// TIA Portal project "WaterFiltering" (V15)

(* hardware
DEVICE "S7-1200 station_1"  S7-1200 Station
   slot 0: "Rack_0"  S7-1200 Rack  Rack  V1.0
   slot 1: "PLC_1"  CPU 1214C AC/DC/Rly  6ES7 214-1BG40-0XB0  V4.2
DEVICE "PC-System_1"  SIMATIC PC station
   slot 0: "SIMATIC PC station"  Rail  SIMATIC PC-Station  V1.0
      slot 125: "Stationmanager"  Station_Manager  V6.0.4
   slot 1: "HMI_RT_1"  WinCC RT Professional  6AV2 105-0xxxx-xxxx  15.0.0.0
   slot 2: "IE general_1"  IE General  IE_CP  V8.2.0
*)

// ===== PLC "PLC_1"  CPU 1214C AC/DC/Rly =====

VAR_GLOBAL   // PLC tag table "Default tag table"
   "FlowSwitch" AT %M0.0 : Bool;
   "PressureInput2" AT %MW0 : Int;
   "PressureInput1" AT %MW2 : Int;
   "ScaledPressure1" AT %MW4 : Int;
   "ScaledPressure2" AT %MW6 : Int;
   "DifferPressureRaw" AT %MW8 : Int;
   "DifferPressure" AT %MW10 : Int;
   "LevelInput" AT %MW12 : Int;
   "ScaledLevel" AT %MW14 : Int;
   "SV1Off_Pb" AT %M16.0 : Bool;
   "SV1Hand_Pb" AT %M16.1 : Bool;
   "SV1Auto_Pb" AT %M16.2 : Bool;
   "SV2Off_Pb" AT %M16.3 : Bool;
   "SV2Hand_Pb" AT %M16.4 : Bool;
   "SV2Auto_pb" AT %M16.5 : Bool;
   "SV3Off_pb" AT %M16.6 : Bool;
   "SV3Hand_pb" AT %M16.7 : Bool;
   "SV3Auto_Pb" AT %M17.0 : Bool;
   "SV4Off_pb" AT %M17.1 : Bool;
   "SV4Hand_Pb" AT %M17.2 : Bool;
   "SV4Auto_Pb" AT %M17.3 : Bool;
   "SV5Off_Pb" AT %M17.4 : Bool;
   "SV5Hand_Pb" AT %M17.5 : Bool;
   "SV5Auto_Pb" AT %M17.6 : Bool;
   "SV6Off_Pb" AT %M17.7 : Bool;
   "SV6Hand_Pb" AT %M18.0 : Bool;
   "SV6Auto_pb" AT %M18.1 : Bool;
   "SV1_Status" AT %MW18 : Int;
   "SV2_Status" AT %MW20 : Int;
   "SV3_Status" AT %MW22 : Int;
   "SV4_Status" AT %MW24 : Int;
   "SV5_Status" AT %MW26 : Int;
   "SV6_Status" AT %MW28 : Int;
   "PumpOff_pb" AT %M2.0 : Bool;
   "PumpHand_pb" AT %M2.1 : Bool;
   "PumpAuto_pb" AT %M2.2 : Bool;
   "Pump_Status" AT %MW30 : Int;
   "AllHOAAuto" AT %M32.0 : Bool;
   "Sys_Running" AT %M32.3 : Bool;
   "Critical_Alarm" AT %M32.6 : Bool;
   "BackWash_Running" AT %M32.7 : Bool;
   "Tank_Filling" AT %M39.0 : Bool;
   "FillStart_Trigger" AT %M33.7 : Bool;
   "FillStop_Trigger" AT %M34.0 : Bool;
   "Alarm_Reset" AT %M34.1 : Bool;
   "HiPresAlarm_Trigger" AT %M34.2 : Bool;
   "HiPres_Alarm" AT %M34.3 : Bool;
   "HiPres_Notify" AT %M34.4 : Bool;
   "Alarm_Silence" AT %M34.5 : Bool;
   "LowFlowAlm_Trigger" AT %M33.0 : Bool;
   "LowFlow_Alarm" AT %M33.1 : Bool;
   "LowAlarm_Notify" AT %M33.2 : Bool;
   "LowLevelAlm_Trigger" AT %M33.3 : Bool;
   "LowLevel_Alarm" AT %M33.4 : Bool;
   "LowLevelAlm_Notify" AT %M33.5 : Bool;
   "HighLevelAlm_Trigger" AT %M34.6 : Bool;
   "HighLevel_Alarm" AT %M34.7 : Bool;
   "HighLevelAlm_notify" AT %M35.0 : Bool;
   "BW_Lockout_Pb" AT %M35.1 : Bool;
   "BW_Lockout" AT %M35.2 : Bool;
   "BW_Enable_Pb" AT %M35.3 : Bool;
   "BWPending_Trigger" AT %M35.4 : Bool;
   "ManualBW_Pb" AT %M35.5 : Bool;
   "BWPending" AT %M35.6 : Bool;
   "BWCycle_Trigger" AT %M35.7 : Bool;
   "BWCount" AT %MW36 : Int;
   "ResetBW_Count_Pb" AT %M38.0 : Bool;
   "Filter_Resistance" AT %MW40 : Int;
   "LowFlowAlm_Pb" AT %M38.1 : Bool;
   "LowFlowAlm_pending" AT %M38.2 : Bool;
   "PutAllIntoAuto" AT %M38.3 : Bool;
   "JustCheck" AT %M38.4 : Bool;
   "St" AT %M38.7 : Bool;
   "FillStart_pulse" AT %M33.6 : Bool;
   "FillStop_Pulse" AT %M39.1 : Bool;
   "SysStart_Pb" AT %M32.1 : Bool;
   "SysStart_Trigger" AT %M32.4 : Bool;
   "SysStop_Pb" AT %M32.5 : Bool;
   "SysStop_Trigger" AT %M38.6 : Bool;
   "SolValve1" AT %Q0.0 : Bool;
   "SolValve2" AT %Q0.1 : Bool;
   "SolValve3" AT %Q0.2 : Bool;
   "SolValve4" AT %Q0.3 : Bool;
   "SolValve5" AT %Q0.4 : Bool;
   "SolValve6" AT %Q0.5 : Bool;
   "Pump" AT %Q0.6 : Bool;
END_VAR

DATA_BLOCK "ALARMS_DB"   // DB1
{ S7_Optimized_Access := 'TRUE' }
VERSION : 0.1
// stored: InstanceOfName ALARMS
"ALARMS"
BEGIN
END_DATA_BLOCK

DATA_BLOCK "MODE_DB"   // DB4
{ S7_Optimized_Access := 'TRUE' }
VERSION : 0.1
// stored: InstanceOfName MODE
"MODE"
BEGIN
END_DATA_BLOCK

DATA_BLOCK "ANALOG_DB"   // DB6
{ S7_Optimized_Access := 'TRUE' }
VERSION : 0.1
// stored: InstanceOfName ANALOG
"ANALOG"
BEGIN
END_DATA_BLOCK

DATA_BLOCK "SIM_DB"   // DB8
{ S7_Optimized_Access := 'TRUE' }
VERSION : 0.1
// stored: InstanceOfName SIM
"SIM"
BEGIN
END_DATA_BLOCK

DATA_BLOCK "LEVEL_DB"   // DB9
{ S7_Optimized_Access := 'TRUE' }
VERSION : 0.1
// stored: InstanceOfName LEVEL
"LEVEL"
BEGIN
END_DATA_BLOCK

DATA_BLOCK "BACKWASH_DB"   // DB10
{ S7_Optimized_Access := 'TRUE' }
VERSION : 0.1
// stored: InstanceOfName BACKWASH
"BACKWASH"
BEGIN
END_DATA_BLOCK

DATA_BLOCK "CTRL_DB"   // DB15
{ S7_Optimized_Access := 'TRUE' }
VERSION : 0.1
// stored: InstanceOfName CTRL
"CTRL"
BEGIN
END_DATA_BLOCK

DATA_BLOCK "HOA_DB"   // DB20
{ S7_Optimized_Access := 'TRUE' }
VERSION : 0.1
// stored: InstanceOfName HOA
"HOA"
BEGIN
END_DATA_BLOCK

DATA_BLOCK "REVIEW_DB"   // DB22
{ S7_Optimized_Access := 'TRUE' }
VERSION : 0.1
// stored: InstanceOfName REVIEW
"REVIEW"
BEGIN
END_DATA_BLOCK

// folder: System blocks/Program resources

DATA_BLOCK "HiPresAlm_Delay"   // DB2
{ S7_Optimized_Access := 'TRUE' }
AUTHOR : Simatic
FAMILY : IEC
NAME : IEC_TMR
VERSION : 1.0
// stored: InstanceOfName IEC_TIMER
"IEC_TIMER"
BEGIN
END_DATA_BLOCK

DATA_BLOCK "LowFlowAlm_Delay"   // DB3
{ S7_Optimized_Access := 'TRUE' }
AUTHOR : Simatic
FAMILY : IEC
NAME : IEC_TMR
VERSION : 1.0
// stored: InstanceOfName IEC_TIMER
"IEC_TIMER"
BEGIN
END_DATA_BLOCK

DATA_BLOCK "FillStart_Delay"   // DB5
{ S7_Optimized_Access := 'TRUE' }
AUTHOR : Simatic
FAMILY : IEC
NAME : IEC_TMR
VERSION : 1.0
// stored: InstanceOfName IEC_TIMER
"IEC_TIMER"
BEGIN
END_DATA_BLOCK

DATA_BLOCK "Simulation_Timer"   // DB7
{ S7_Optimized_Access := 'TRUE' }
AUTHOR : Simatic
FAMILY : IEC
NAME : IEC_TMR
VERSION : 1.0
// stored: InstanceOfName IEC_TIMER
"IEC_TIMER"
BEGIN
END_DATA_BLOCK

DATA_BLOCK "FillStop_Delay"   // DB11
{ S7_Optimized_Access := 'TRUE' }
AUTHOR : Simatic
FAMILY : IEC
NAME : IEC_TMR
VERSION : 1.0
// stored: InstanceOfName IEC_TIMER
"IEC_TIMER"
BEGIN
END_DATA_BLOCK

DATA_BLOCK "HiLevelAlm_Delay"   // DB13
{ S7_Optimized_Access := 'TRUE' }
AUTHOR : Simatic
FAMILY : IEC
NAME : IEC_TMR
VERSION : 1.0
// stored: InstanceOfName IEC_TIMER
"IEC_TIMER"
BEGIN
END_DATA_BLOCK

DATA_BLOCK "LowLevelAlm_Delay"   // DB14
{ S7_Optimized_Access := 'TRUE' }
AUTHOR : Simatic
FAMILY : IEC
NAME : IEC_TMR
VERSION : 1.0
// stored: InstanceOfName IEC_TIMER
"IEC_TIMER"
BEGIN
END_DATA_BLOCK

DATA_BLOCK "BWPending_Delay"   // DB16
{ S7_Optimized_Access := 'TRUE' }
AUTHOR : Simatic
FAMILY : IEC
NAME : IEC_TMR
VERSION : 1.0
// stored: InstanceOfName IEC_TIMER
"IEC_TIMER"
BEGIN
END_DATA_BLOCK

DATA_BLOCK "BWCycle_Delay"   // DB17
{ S7_Optimized_Access := 'TRUE' }
AUTHOR : Simatic
FAMILY : IEC
NAME : IEC_TMR
VERSION : 1.0
// stored: InstanceOfName IEC_TIMER
"IEC_TIMER"
BEGIN
END_DATA_BLOCK

DATA_BLOCK "BWCycle"   // DB18
{ S7_Optimized_Access := 'TRUE' }
AUTHOR : Simatic
FAMILY : IEC
NAME : IEC_TMR
VERSION : 1.0
// stored: InstanceOfName IEC_TIMER
"IEC_TIMER"
BEGIN
END_DATA_BLOCK

DATA_BLOCK "ResetBWCount_Delay"   // DB19
{ S7_Optimized_Access := 'TRUE' }
AUTHOR : Simatic
FAMILY : IEC
NAME : IEC_TMR
VERSION : 1.0
// stored: InstanceOfName IEC_TIMER
"IEC_TIMER"
BEGIN
END_DATA_BLOCK

DATA_BLOCK "FlowSWClose_Delay"   // DB21
{ S7_Optimized_Access := 'TRUE' }
AUTHOR : Simatic
FAMILY : IEC
NAME : IEC_TMR
VERSION : 1.0
// stored: InstanceOfName IEC_TIMER
"IEC_TIMER"
BEGIN
END_DATA_BLOCK

// folder: (top level)

FUNCTION_BLOCK "ANALOG"   // FB1, LAD
{ S7_Optimized_Access := 'TRUE' }
VERSION : 0.1
BEGIN

REGION Network 1
   // Analog Input : Pressure(0-20 psi), Water level(0-100)
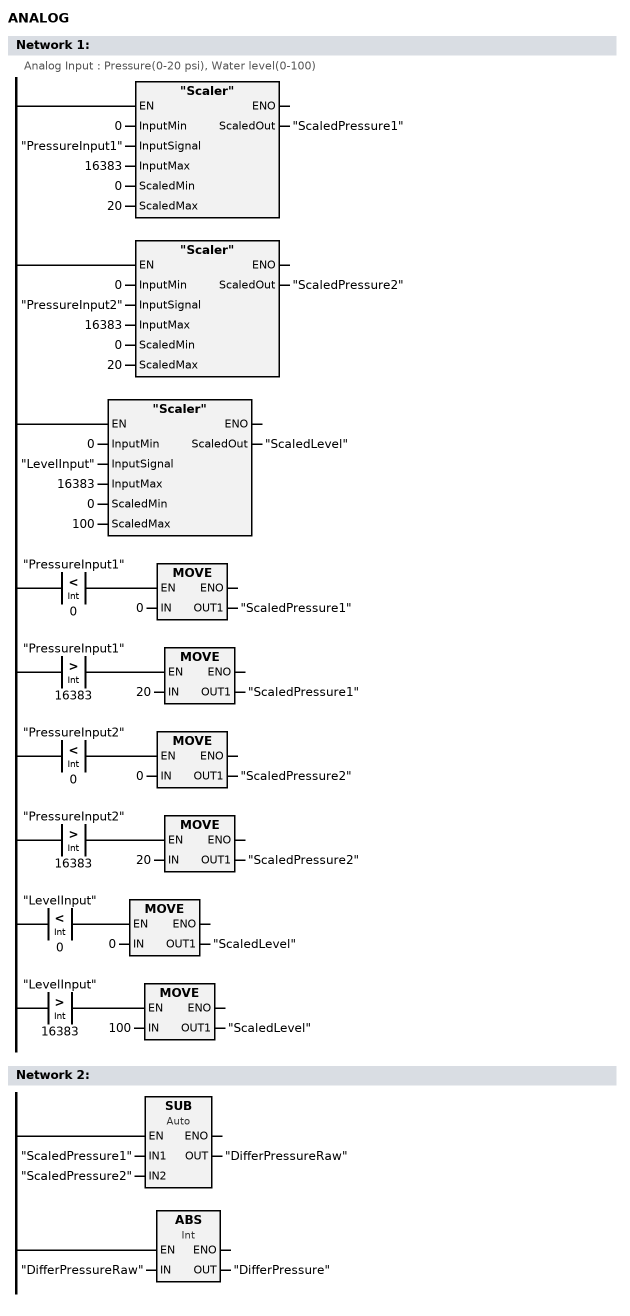
   RUNG wire#powerrail
      "Scaler"(InputMin := 0, InputSignal := "PressureInput1", InputMax := 16383, ScaledMin := 0, ScaledMax := 20, ScaledOut => "ScaledPressure1")
   END_RUNG
   RUNG wire#powerrail
      "Scaler"(InputMin := 0, InputSignal := "PressureInput2", InputMax := 16383, ScaledMin := 0, ScaledMax := 20, ScaledOut => "ScaledPressure2")
   END_RUNG
   RUNG wire#powerrail
      "Scaler"(InputMin := 0, InputSignal := "LevelInput", InputMax := 16383, ScaledMin := 0, ScaledMax := 100, ScaledOut => "ScaledLevel")
   END_RUNG
   RUNG wire#powerrail
      { S7_Templates := "SrcType := Int" } LT_Contact(in1 := "PressureInput1", in2 := 0)
      { S7_GenerateENO := "TRUE" } Move(in := 0, out1 => "ScaledPressure1")
   END_RUNG
   RUNG wire#powerrail
      { S7_Templates := "SrcType := Int" } GT_Contact(in1 := "PressureInput1", in2 := 16383)
      { S7_GenerateENO := "TRUE" } Move(in := 20, out1 => "ScaledPressure1")
   END_RUNG
   RUNG wire#powerrail
      { S7_Templates := "SrcType := Int" } LT_Contact(in1 := "PressureInput2", in2 := 0)
      { S7_GenerateENO := "TRUE" } Move(in := 0, out1 => "ScaledPressure2")
   END_RUNG
   RUNG wire#powerrail
      { S7_Templates := "SrcType := Int" } GT_Contact(in1 := "PressureInput2", in2 := 16383)
      { S7_GenerateENO := "TRUE" } Move(in := 20, out1 => "ScaledPressure2")
   END_RUNG
   RUNG wire#powerrail
      { S7_Templates := "SrcType := Int" } LT_Contact(in1 := "LevelInput", in2 := 0)
      { S7_GenerateENO := "TRUE" } Move(in := 0, out1 => "ScaledLevel")
   END_RUNG
   RUNG wire#powerrail
      { S7_Templates := "SrcType := Int" } GT_Contact(in1 := "LevelInput", in2 := 16383)
      { S7_GenerateENO := "TRUE" } Move(in := 100, out1 => "ScaledLevel")
   END_RUNG
   // the same network as SCL:
   "Scaler"(InputMin := 0,
            InputSignal := "PressureInput1",
            InputMax := 16383,
            ScaledMin := 0,
            ScaledMax := 20,
            ScaledOut => "ScaledPressure1");
   "Scaler"(InputMin := 0,
            InputSignal := "PressureInput2",
            InputMax := 16383,
            ScaledMin := 0,
            ScaledMax := 20,
            ScaledOut => "ScaledPressure2");
   "Scaler"(InputMin := 0,
            InputSignal := "LevelInput",
            InputMax := 16383,
            ScaledMin := 0,
            ScaledMax := 100,
            ScaledOut => "ScaledLevel");
   IF "PressureInput1" < 0 THEN "ScaledPressure1" := 0; END_IF;
   IF "PressureInput1" > 16383 THEN "ScaledPressure1" := 20; END_IF;
   IF "PressureInput2" < 0 THEN "ScaledPressure2" := 0; END_IF;
   IF "PressureInput2" > 16383 THEN "ScaledPressure2" := 20; END_IF;
   IF "LevelInput" < 0 THEN "ScaledLevel" := 0; END_IF;
   IF "LevelInput" > 16383 THEN "ScaledLevel" := 100; END_IF;
END_REGION

REGION Network 2
   RUNG wire#powerrail
      { S7_GenerateENO := "TRUE" } Sub(in1 := "ScaledPressure1", in2 := "ScaledPressure2", out => "DifferPressureRaw")
   END_RUNG
   RUNG wire#powerrail
      { S7_Templates := "SrcType := Int"; S7_GenerateENO := "TRUE" } Abs(in := "DifferPressureRaw", out => "DifferPressure")
   END_RUNG
   // the same network as SCL:
   "DifferPressureRaw" := "ScaledPressure1" - "ScaledPressure2";
   "DifferPressure" := ABS("DifferPressureRaw");
END_REGION
END_FUNCTION_BLOCK

FUNCTION_BLOCK "ALARMS"   // FB2, LAD
{ S7_Optimized_Access := 'TRUE' }
VERSION : 0.1
   VAR
      ons1 : Bool;
      ons2 : Bool;
      ons3 : Bool;
      ons4 : Bool;
   END_VAR
   VAR_TEMP   // added for the SCL form of the ladder/FBD networks
      _w1 : Bool;
   END_VAR
BEGIN

REGION Network 1
   // High Pressure Alarm
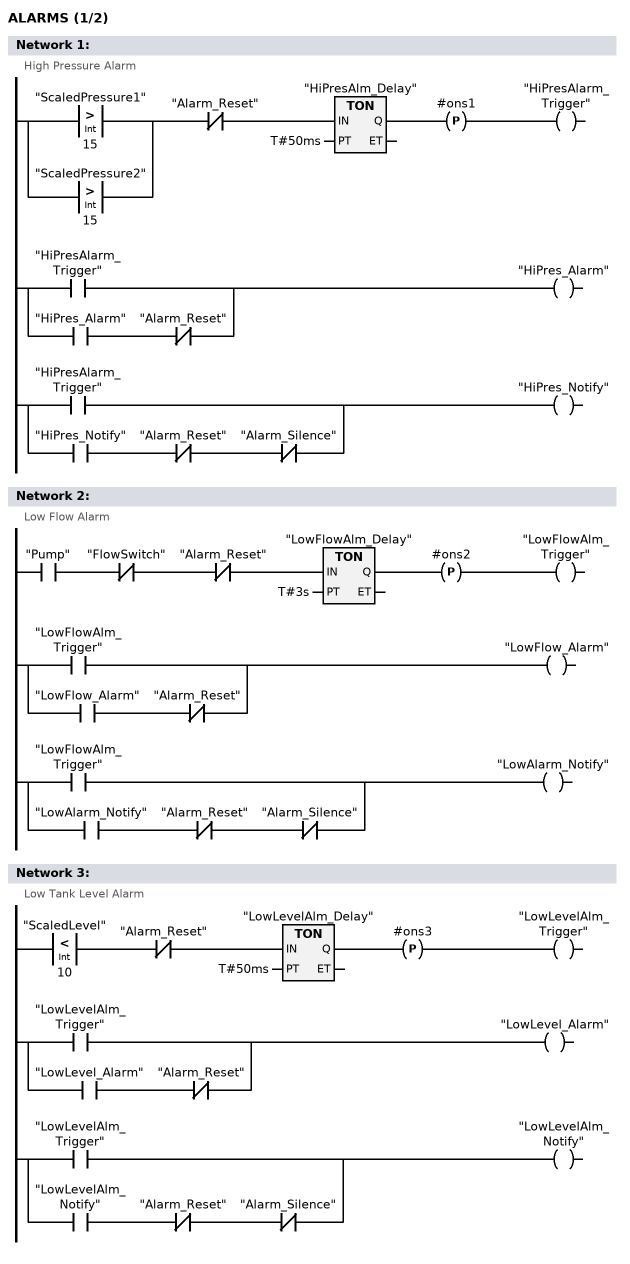
   "HiPresAlm_Delay".TON(IN := (("ScaledPressure1" > 15) OR ("ScaledPressure2" > 15)) AND NOT "Alarm_Reset",
                         PT := T#50ms);
   #_w1 := "HiPresAlm_Delay".Q AND NOT #ons1;   // rising edge
   #ons1 := "HiPresAlm_Delay".Q;
   "HiPresAlarm_Trigger" := #_w1;
   "HiPres_Alarm" := "HiPresAlarm_Trigger" OR ("HiPres_Alarm" AND NOT "Alarm_Reset");
   "HiPres_Notify" := "HiPresAlarm_Trigger" OR ("HiPres_Notify" AND NOT "Alarm_Reset" AND NOT "Alarm_Silence");
END_REGION

REGION Network 2
   // Low Flow Alarm
   "LowFlowAlm_Delay".TON(IN := "Pump" AND NOT "FlowSwitch" AND NOT "Alarm_Reset", PT := T#3s);
   #_w1 := "LowFlowAlm_Delay".Q AND NOT #ons2;   // rising edge
   #ons2 := "LowFlowAlm_Delay".Q;
   "LowFlowAlm_Trigger" := #_w1;
   "LowFlow_Alarm" := "LowFlowAlm_Trigger" OR ("LowFlow_Alarm" AND NOT "Alarm_Reset");
   "LowAlarm_Notify" := "LowFlowAlm_Trigger" OR ("LowAlarm_Notify" AND NOT "Alarm_Reset" AND NOT "Alarm_Silence");
END_REGION

REGION Network 3
   // Low Tank Level Alarm
   "LowLevelAlm_Delay".TON(IN := ("ScaledLevel" < 10) AND NOT "Alarm_Reset", PT := T#50ms);
   #_w1 := "LowLevelAlm_Delay".Q AND NOT #ons3;   // rising edge
   #ons3 := "LowLevelAlm_Delay".Q;
   "LowLevelAlm_Trigger" := #_w1;
   "LowLevel_Alarm" := "LowLevelAlm_Trigger" OR ("LowLevel_Alarm" AND NOT "Alarm_Reset");
   "LowLevelAlm_Notify" := "LowLevelAlm_Trigger" OR ("LowLevelAlm_Notify" AND NOT "Alarm_Reset" AND NOT "Alarm_Silence");
END_REGION

REGION Network 4
   // High Level Alarm
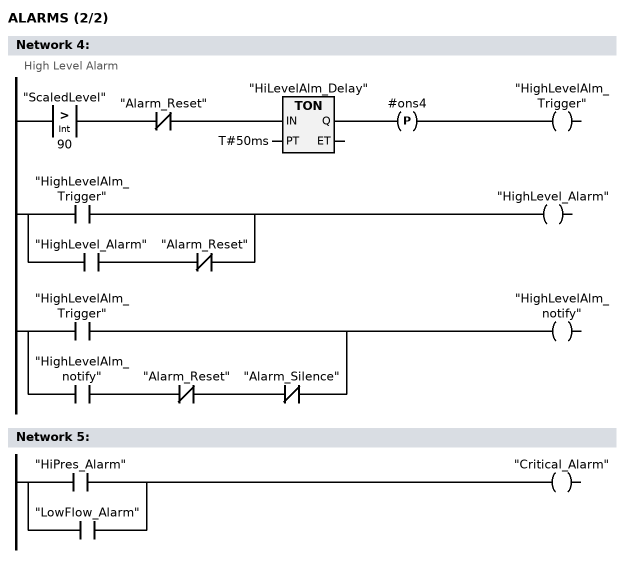
   "HiLevelAlm_Delay".TON(IN := ("ScaledLevel" > 90) AND NOT "Alarm_Reset", PT := T#50ms);
   #_w1 := "HiLevelAlm_Delay".Q AND NOT #ons4;   // rising edge
   #ons4 := "HiLevelAlm_Delay".Q;
   "HighLevelAlm_Trigger" := #_w1;
   "HighLevel_Alarm" := "HighLevelAlm_Trigger" OR ("HighLevel_Alarm" AND NOT "Alarm_Reset");
   "HighLevelAlm_notify" := "HighLevelAlm_Trigger" OR ("HighLevelAlm_notify" AND NOT "Alarm_Reset" AND NOT "Alarm_Silence");
END_REGION

REGION Network 5
   RUNG wire#powerrail
      Contact( "HiPres_Alarm" )
      wire#w1
      Coil( "Critical_Alarm" )
   END_RUNG
   RUNG wire#powerrail
      Contact( "LowFlow_Alarm" )
   END_RUNG wire#w1
   // the same network as SCL:
   "Critical_Alarm" := "HiPres_Alarm" OR "LowFlow_Alarm";
END_REGION
END_FUNCTION_BLOCK

FUNCTION_BLOCK "CTRL"   // FB3, LAD
{ S7_Optimized_Access := 'TRUE' }
VERSION : 0.1
BEGIN

REGION Network 1
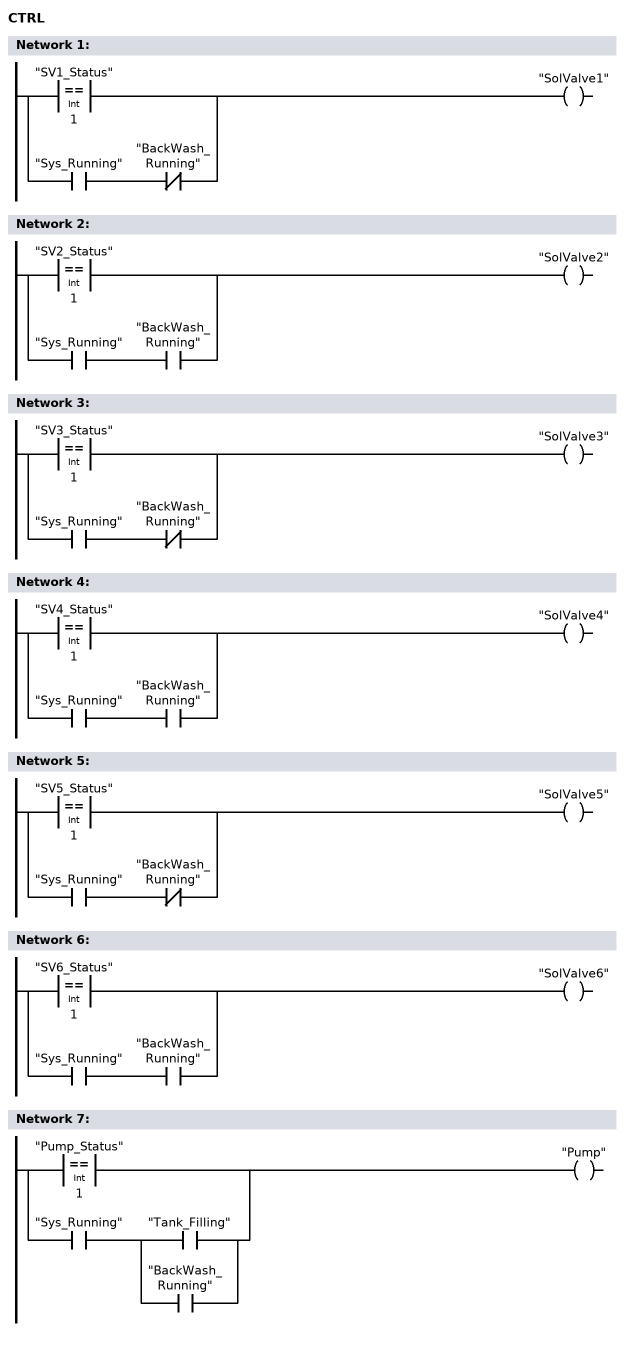
   RUNG wire#powerrail
      { S7_Templates := "SrcType := Int" } EQ_Contact(in1 := "SV1_Status", in2 := 1)
      wire#w1
      Coil( "SolValve1" )
   END_RUNG
   RUNG wire#powerrail
      Contact( "Sys_Running" )
      I_Contact( "BackWash_Running" )
   END_RUNG wire#w1
   // the same network as SCL:
   "SolValve1" := ("SV1_Status" = 1) OR ("Sys_Running" AND NOT "BackWash_Running");
END_REGION

REGION Network 2
   RUNG wire#powerrail
      { S7_Templates := "SrcType := Int" } EQ_Contact(in1 := "SV2_Status", in2 := 1)
      wire#w1
      Coil( "SolValve2" )
   END_RUNG
   RUNG wire#powerrail
      Contact( "Sys_Running" )
      Contact( "BackWash_Running" )
   END_RUNG wire#w1
   // the same network as SCL:
   "SolValve2" := ("SV2_Status" = 1) OR ("Sys_Running" AND "BackWash_Running");
END_REGION

REGION Network 3
   RUNG wire#powerrail
      { S7_Templates := "SrcType := Int" } EQ_Contact(in1 := "SV3_Status", in2 := 1)
      wire#w1
      Coil( "SolValve3" )
   END_RUNG
   RUNG wire#powerrail
      Contact( "Sys_Running" )
      I_Contact( "BackWash_Running" )
   END_RUNG wire#w1
   // the same network as SCL:
   "SolValve3" := ("SV3_Status" = 1) OR ("Sys_Running" AND NOT "BackWash_Running");
END_REGION

REGION Network 4
   RUNG wire#powerrail
      { S7_Templates := "SrcType := Int" } EQ_Contact(in1 := "SV4_Status", in2 := 1)
      wire#w1
      Coil( "SolValve4" )
   END_RUNG
   RUNG wire#powerrail
      Contact( "Sys_Running" )
      Contact( "BackWash_Running" )
   END_RUNG wire#w1
   // the same network as SCL:
   "SolValve4" := ("SV4_Status" = 1) OR ("Sys_Running" AND "BackWash_Running");
END_REGION

REGION Network 5
   RUNG wire#powerrail
      { S7_Templates := "SrcType := Int" } EQ_Contact(in1 := "SV5_Status", in2 := 1)
      wire#w1
      Coil( "SolValve5" )
   END_RUNG
   RUNG wire#powerrail
      Contact( "Sys_Running" )
      I_Contact( "BackWash_Running" )
   END_RUNG wire#w1
   // the same network as SCL:
   "SolValve5" := ("SV5_Status" = 1) OR ("Sys_Running" AND NOT "BackWash_Running");
END_REGION

REGION Network 6
   RUNG wire#powerrail
      { S7_Templates := "SrcType := Int" } EQ_Contact(in1 := "SV6_Status", in2 := 1)
      wire#w1
      Coil( "SolValve6" )
   END_RUNG
   RUNG wire#powerrail
      Contact( "Sys_Running" )
      Contact( "BackWash_Running" )
   END_RUNG wire#w1
   // the same network as SCL:
   "SolValve6" := ("SV6_Status" = 1) OR ("Sys_Running" AND "BackWash_Running");
END_REGION

REGION Network 7
   RUNG wire#powerrail
      { S7_Templates := "SrcType := Int" } EQ_Contact(in1 := "Pump_Status", in2 := 1)
      wire#w1
      Coil( "Pump" )
   END_RUNG
   RUNG wire#powerrail
      Contact( "Sys_Running" )
      wire#w2
      Contact( "Tank_Filling" )
   END_RUNG wire#w1
   RUNG wire#w2
      Contact( "BackWash_Running" )
   END_RUNG wire#w1
   // the same network as SCL:
   "Pump" := ("Pump_Status" = 1) OR ("Sys_Running" AND ("Tank_Filling" OR "BackWash_Running"));
END_REGION
END_FUNCTION_BLOCK

FUNCTION_BLOCK "HOA"   // FB4, LAD
{ S7_Optimized_Access := 'TRUE' }
VERSION : 0.1
   VAR
      ons1 : Bool;
      ons2 : Bool;
      ons3 : Bool;
      ons4 : Bool;
      ons5 : Bool;
      ons6 : Bool;
      ons7 : Bool;
      ons8 : Bool;
      ons9 : Bool;
      ons10 : Bool;
      ons11 : Bool;
      ons12 : Bool;
      ons13 : Bool;
      ons14 : Bool;
      ons15 : Bool;
      ons16 : Bool;
      ons17 : Bool;
      ons18 : Bool;
      ons19 : Bool;
      ons20 : Bool;
      ons21 : Bool;
   END_VAR
   VAR_TEMP   // added for the SCL form of the ladder/FBD networks
      _w1 : Bool;
      _w2 : Bool;
      _w3 : Bool;
   END_VAR
BEGIN

REGION Network 1
   // Solenoid Valve1 HOA
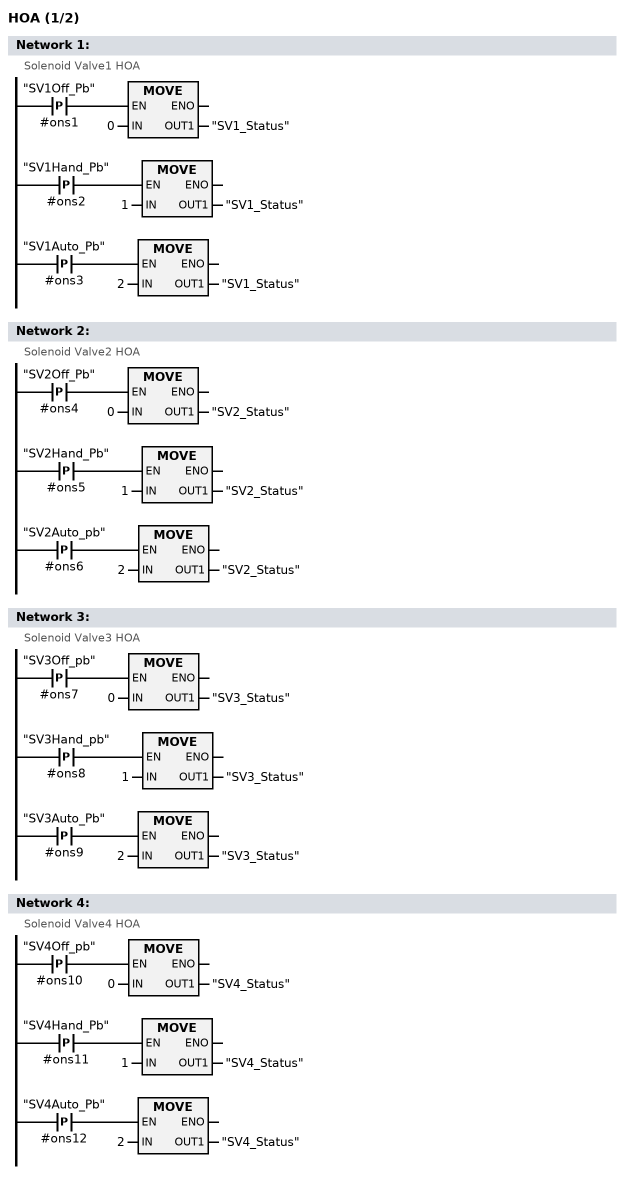
   RUNG wire#powerrail
      P_Contact(operand := "SV1Off_Pb", bit := #ons1)
      { S7_GenerateENO := "TRUE" } Move(in := 0, out1 => "SV1_Status")
   END_RUNG
   RUNG wire#powerrail
      P_Contact(operand := "SV1Hand_Pb", bit := #ons2)
      { S7_GenerateENO := "TRUE" } Move(in := 1, out1 => "SV1_Status")
   END_RUNG
   RUNG wire#powerrail
      P_Contact(operand := "SV1Auto_Pb", bit := #ons3)
      { S7_GenerateENO := "TRUE" } Move(in := 2, out1 => "SV1_Status")
   END_RUNG
   // the same network as SCL:
   #_w1 := "SV1Off_Pb" AND NOT #ons1;   // rising edge of "SV1Off_Pb"
   #ons1 := "SV1Off_Pb";
   IF #_w1 THEN "SV1_Status" := 0; END_IF;
   #_w2 := "SV1Hand_Pb" AND NOT #ons2;   // rising edge of "SV1Hand_Pb"
   #ons2 := "SV1Hand_Pb";
   IF #_w2 THEN "SV1_Status" := 1; END_IF;
   #_w3 := "SV1Auto_Pb" AND NOT #ons3;   // rising edge of "SV1Auto_Pb"
   #ons3 := "SV1Auto_Pb";
   IF #_w3 THEN "SV1_Status" := 2; END_IF;
END_REGION

REGION Network 2
   // Solenoid Valve2 HOA
   RUNG wire#powerrail
      P_Contact(operand := "SV2Off_Pb", bit := #ons4)
      { S7_GenerateENO := "TRUE" } Move(in := 0, out1 => "SV2_Status")
   END_RUNG
   RUNG wire#powerrail
      P_Contact(operand := "SV2Hand_Pb", bit := #ons5)
      { S7_GenerateENO := "TRUE" } Move(in := 1, out1 => "SV2_Status")
   END_RUNG
   RUNG wire#powerrail
      P_Contact(operand := "SV2Auto_pb", bit := #ons6)
      { S7_GenerateENO := "TRUE" } Move(in := 2, out1 => "SV2_Status")
   END_RUNG
   // the same network as SCL:
   #_w1 := "SV2Off_Pb" AND NOT #ons4;   // rising edge of "SV2Off_Pb"
   #ons4 := "SV2Off_Pb";
   IF #_w1 THEN "SV2_Status" := 0; END_IF;
   #_w2 := "SV2Hand_Pb" AND NOT #ons5;   // rising edge of "SV2Hand_Pb"
   #ons5 := "SV2Hand_Pb";
   IF #_w2 THEN "SV2_Status" := 1; END_IF;
   #_w3 := "SV2Auto_pb" AND NOT #ons6;   // rising edge of "SV2Auto_pb"
   #ons6 := "SV2Auto_pb";
   IF #_w3 THEN "SV2_Status" := 2; END_IF;
END_REGION

REGION Network 3
   // Solenoid Valve3 HOA
   RUNG wire#powerrail
      P_Contact(operand := "SV3Off_pb", bit := #ons7)
      { S7_GenerateENO := "TRUE" } Move(in := 0, out1 => "SV3_Status")
   END_RUNG
   RUNG wire#powerrail
      P_Contact(operand := "SV3Hand_pb", bit := #ons8)
      { S7_GenerateENO := "TRUE" } Move(in := 1, out1 => "SV3_Status")
   END_RUNG
   RUNG wire#powerrail
      P_Contact(operand := "SV3Auto_Pb", bit := #ons9)
      { S7_GenerateENO := "TRUE" } Move(in := 2, out1 => "SV3_Status")
   END_RUNG
   // the same network as SCL:
   #_w1 := "SV3Off_pb" AND NOT #ons7;   // rising edge of "SV3Off_pb"
   #ons7 := "SV3Off_pb";
   IF #_w1 THEN "SV3_Status" := 0; END_IF;
   #_w2 := "SV3Hand_pb" AND NOT #ons8;   // rising edge of "SV3Hand_pb"
   #ons8 := "SV3Hand_pb";
   IF #_w2 THEN "SV3_Status" := 1; END_IF;
   #_w3 := "SV3Auto_Pb" AND NOT #ons9;   // rising edge of "SV3Auto_Pb"
   #ons9 := "SV3Auto_Pb";
   IF #_w3 THEN "SV3_Status" := 2; END_IF;
END_REGION

REGION Network 4
   // Solenoid Valve4 HOA
   RUNG wire#powerrail
      P_Contact(operand := "SV4Off_pb", bit := #ons10)
      { S7_GenerateENO := "TRUE" } Move(in := 0, out1 => "SV4_Status")
   END_RUNG
   RUNG wire#powerrail
      P_Contact(operand := "SV4Hand_Pb", bit := #ons11)
      { S7_GenerateENO := "TRUE" } Move(in := 1, out1 => "SV4_Status")
   END_RUNG
   RUNG wire#powerrail
      P_Contact(operand := "SV4Auto_Pb", bit := #ons12)
      { S7_GenerateENO := "TRUE" } Move(in := 2, out1 => "SV4_Status")
   END_RUNG
   // the same network as SCL:
   #_w1 := "SV4Off_pb" AND NOT #ons10;   // rising edge of "SV4Off_pb"
   #ons10 := "SV4Off_pb";
   IF #_w1 THEN "SV4_Status" := 0; END_IF;
   #_w2 := "SV4Hand_Pb" AND NOT #ons11;   // rising edge of "SV4Hand_Pb"
   #ons11 := "SV4Hand_Pb";
   IF #_w2 THEN "SV4_Status" := 1; END_IF;
   #_w3 := "SV4Auto_Pb" AND NOT #ons12;   // rising edge of "SV4Auto_Pb"
   #ons12 := "SV4Auto_Pb";
   IF #_w3 THEN "SV4_Status" := 2; END_IF;
END_REGION

REGION Network 5
   // Solenoid Valve5 HOA
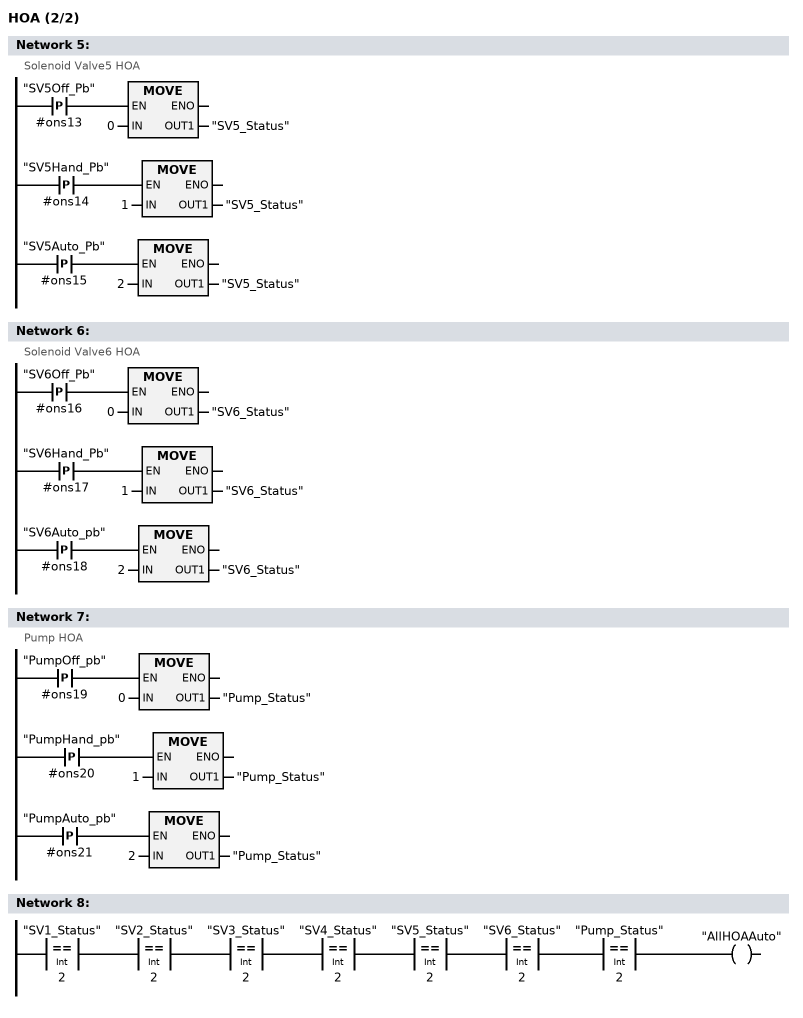
   RUNG wire#powerrail
      P_Contact(operand := "SV5Off_Pb", bit := #ons13)
      { S7_GenerateENO := "TRUE" } Move(in := 0, out1 => "SV5_Status")
   END_RUNG
   RUNG wire#powerrail
      P_Contact(operand := "SV5Hand_Pb", bit := #ons14)
      { S7_GenerateENO := "TRUE" } Move(in := 1, out1 => "SV5_Status")
   END_RUNG
   RUNG wire#powerrail
      P_Contact(operand := "SV5Auto_Pb", bit := #ons15)
      { S7_GenerateENO := "TRUE" } Move(in := 2, out1 => "SV5_Status")
   END_RUNG
   // the same network as SCL:
   #_w1 := "SV5Off_Pb" AND NOT #ons13;   // rising edge of "SV5Off_Pb"
   #ons13 := "SV5Off_Pb";
   IF #_w1 THEN "SV5_Status" := 0; END_IF;
   #_w2 := "SV5Hand_Pb" AND NOT #ons14;   // rising edge of "SV5Hand_Pb"
   #ons14 := "SV5Hand_Pb";
   IF #_w2 THEN "SV5_Status" := 1; END_IF;
   #_w3 := "SV5Auto_Pb" AND NOT #ons15;   // rising edge of "SV5Auto_Pb"
   #ons15 := "SV5Auto_Pb";
   IF #_w3 THEN "SV5_Status" := 2; END_IF;
END_REGION

REGION Network 6
   // Solenoid Valve6 HOA
   RUNG wire#powerrail
      P_Contact(operand := "SV6Off_Pb", bit := #ons16)
      { S7_GenerateENO := "TRUE" } Move(in := 0, out1 => "SV6_Status")
   END_RUNG
   RUNG wire#powerrail
      P_Contact(operand := "SV6Hand_Pb", bit := #ons17)
      { S7_GenerateENO := "TRUE" } Move(in := 1, out1 => "SV6_Status")
   END_RUNG
   RUNG wire#powerrail
      P_Contact(operand := "SV6Auto_pb", bit := #ons18)
      { S7_GenerateENO := "TRUE" } Move(in := 2, out1 => "SV6_Status")
   END_RUNG
   // the same network as SCL:
   #_w1 := "SV6Off_Pb" AND NOT #ons16;   // rising edge of "SV6Off_Pb"
   #ons16 := "SV6Off_Pb";
   IF #_w1 THEN "SV6_Status" := 0; END_IF;
   #_w2 := "SV6Hand_Pb" AND NOT #ons17;   // rising edge of "SV6Hand_Pb"
   #ons17 := "SV6Hand_Pb";
   IF #_w2 THEN "SV6_Status" := 1; END_IF;
   #_w3 := "SV6Auto_pb" AND NOT #ons18;   // rising edge of "SV6Auto_pb"
   #ons18 := "SV6Auto_pb";
   IF #_w3 THEN "SV6_Status" := 2; END_IF;
END_REGION

REGION Network 7
   // Pump HOA
   RUNG wire#powerrail
      P_Contact(operand := "PumpOff_pb", bit := #ons19)
      { S7_GenerateENO := "TRUE" } Move(in := 0, out1 => "Pump_Status")
   END_RUNG
   RUNG wire#powerrail
      P_Contact(operand := "PumpHand_pb", bit := #ons20)
      { S7_GenerateENO := "TRUE" } Move(in := 1, out1 => "Pump_Status")
   END_RUNG
   RUNG wire#powerrail
      P_Contact(operand := "PumpAuto_pb", bit := #ons21)
      { S7_GenerateENO := "TRUE" } Move(in := 2, out1 => "Pump_Status")
   END_RUNG
   // the same network as SCL:
   #_w1 := "PumpOff_pb" AND NOT #ons19;   // rising edge of "PumpOff_pb"
   #ons19 := "PumpOff_pb";
   IF #_w1 THEN "Pump_Status" := 0; END_IF;
   #_w2 := "PumpHand_pb" AND NOT #ons20;   // rising edge of "PumpHand_pb"
   #ons20 := "PumpHand_pb";
   IF #_w2 THEN "Pump_Status" := 1; END_IF;
   #_w3 := "PumpAuto_pb" AND NOT #ons21;   // rising edge of "PumpAuto_pb"
   #ons21 := "PumpAuto_pb";
   IF #_w3 THEN "Pump_Status" := 2; END_IF;
END_REGION

REGION Network 8
   RUNG wire#powerrail
      { S7_Templates := "SrcType := Int" } EQ_Contact(in1 := "SV1_Status", in2 := 2)
      { S7_Templates := "SrcType := Int" } EQ_Contact(in1 := "SV2_Status", in2 := 2)
      { S7_Templates := "SrcType := Int" } EQ_Contact(in1 := "SV3_Status", in2 := 2)
      { S7_Templates := "SrcType := Int" } EQ_Contact(in1 := "SV4_Status", in2 := 2)
      { S7_Templates := "SrcType := Int" } EQ_Contact(in1 := "SV5_Status", in2 := 2)
      { S7_Templates := "SrcType := Int" } EQ_Contact(in1 := "SV6_Status", in2 := 2)
      { S7_Templates := "SrcType := Int" } EQ_Contact(in1 := "Pump_Status", in2 := 2)
      Coil( "AllHOAAuto" )
   END_RUNG
   // the same network as SCL:
   "AllHOAAuto" := ("SV1_Status" = 2) AND ("SV2_Status" = 2) AND ("SV3_Status" = 2) AND ("SV4_Status" = 2) AND ("SV5_Status" = 2) AND ("SV6_Status" = 2) AND ("Pump_Status" = 2);
END_REGION
END_FUNCTION_BLOCK

FUNCTION_BLOCK "SIM"   // FB5, LAD
{ S7_Optimized_Access := 'TRUE' }
VERSION : 0.1
BEGIN

REGION Network 1
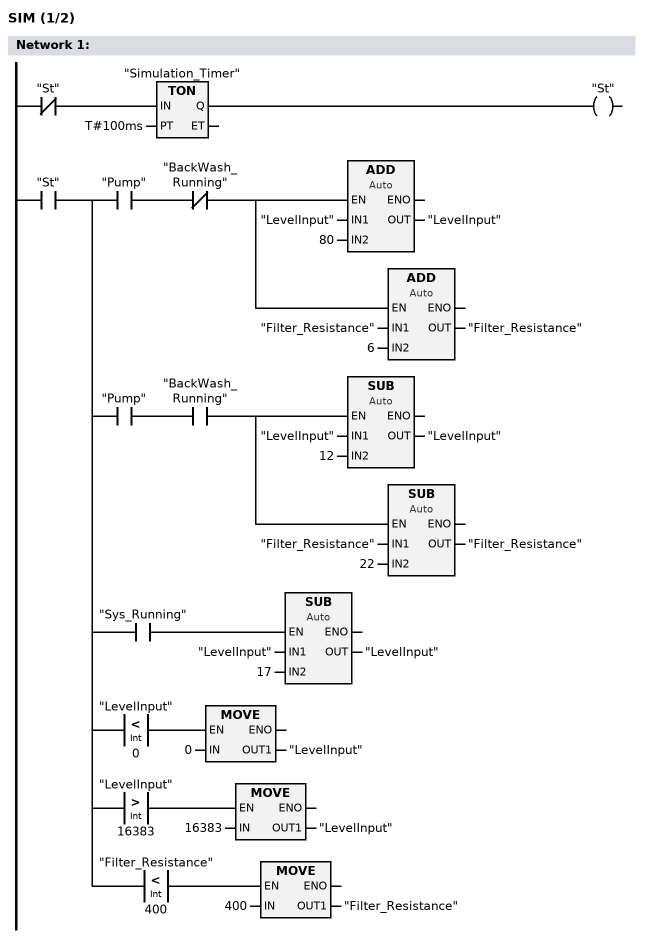
   "Simulation_Timer".TON(IN := NOT "St", PT := T#100ms);
   "St" := "Simulation_Timer".Q;
   IF "St" AND "Pump" AND NOT "BackWash_Running" THEN
       "LevelInput" := "LevelInput" + 80;
       "Filter_Resistance" := "Filter_Resistance" + 6;
   END_IF;
   IF "St" AND "Pump" AND "BackWash_Running" THEN
       "LevelInput" := "LevelInput" - 12;
       "Filter_Resistance" := "Filter_Resistance" - 22;
   END_IF;
   IF "St" AND "Sys_Running" THEN "LevelInput" := "LevelInput" - 17; END_IF;
   IF "St" AND ("LevelInput" < 0) THEN "LevelInput" := 0; END_IF;
   IF "St" AND ("LevelInput" > 16383) THEN "LevelInput" := 16383; END_IF;
   IF "St" AND ("Filter_Resistance" < 400) THEN "Filter_Resistance" := 400; END_IF;
END_REGION

REGION Network 2
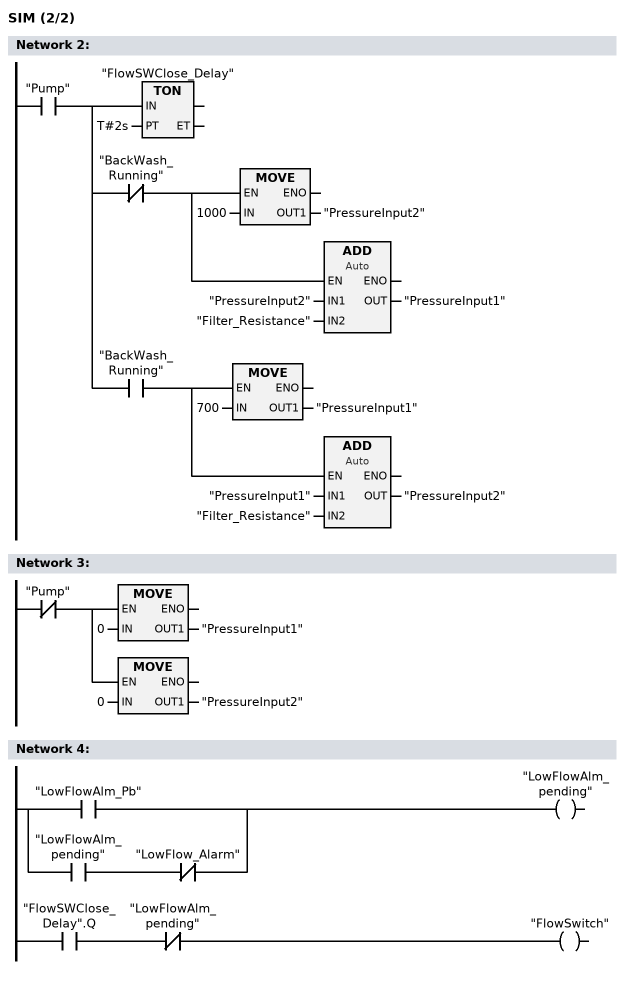
   "FlowSWClose_Delay".TON(IN := "Pump", PT := T#2s);
   IF "Pump" AND NOT "BackWash_Running" THEN
       "PressureInput2" := 1000;
       "PressureInput1" := "PressureInput2" + "Filter_Resistance";
   END_IF;
   IF "Pump" AND "BackWash_Running" THEN
       "PressureInput1" := 700;
       "PressureInput2" := "PressureInput1" + "Filter_Resistance";
   END_IF;
END_REGION

REGION Network 3
   RUNG wire#powerrail
      I_Contact( "Pump" )
      wire#w1
      { S7_GenerateENO := "TRUE" } Move(in := 0, out1 => "PressureInput1")
   END_RUNG
   RUNG wire#w1
      { S7_GenerateENO := "TRUE" } Move(in := 0, out1 => "PressureInput2")
   END_RUNG
   // the same network as SCL:
   IF NOT "Pump" THEN
       "PressureInput1" := 0;
       "PressureInput2" := 0;
   END_IF;
END_REGION

REGION Network 4
   RUNG wire#powerrail
      Contact( "LowFlowAlm_Pb" )
      wire#w1
      Coil( "LowFlowAlm_pending" )
   END_RUNG
   RUNG wire#powerrail
      Contact( "LowFlowAlm_pending" )
      I_Contact( "LowFlow_Alarm" )
   END_RUNG wire#w1
   RUNG wire#powerrail
      Contact( "FlowSWClose_Delay".Q )
      I_Contact( "LowFlowAlm_pending" )
      Coil( "FlowSwitch" )
   END_RUNG
   // the same network as SCL:
   "LowFlowAlm_pending" := "LowFlowAlm_Pb" OR ("LowFlowAlm_pending" AND NOT "LowFlow_Alarm");
   "FlowSwitch" := "FlowSWClose_Delay".Q AND NOT "LowFlowAlm_pending";
END_REGION
END_FUNCTION_BLOCK

FUNCTION_BLOCK "MODE"   // FB6, LAD
{ S7_Optimized_Access := 'TRUE' }
VERSION : 0.1
   VAR
      ons1 : Bool;
      ons2 : Bool;
   END_VAR
BEGIN

REGION Network 1
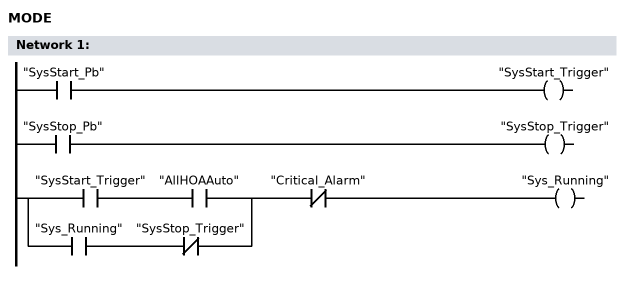
   RUNG wire#powerrail
      Contact( "SysStart_Pb" )
      Coil( "SysStart_Trigger" )
   END_RUNG
   RUNG wire#powerrail
      Contact( "SysStop_Pb" )
      Coil( "SysStop_Trigger" )
   END_RUNG
   RUNG wire#powerrail
      Contact( "SysStart_Trigger" )
      Contact( "AllHOAAuto" )
      wire#w1
      I_Contact( "Critical_Alarm" )
      Coil( "Sys_Running" )
   END_RUNG
   RUNG wire#powerrail
      Contact( "Sys_Running" )
      I_Contact( "SysStop_Trigger" )
   END_RUNG wire#w1
   // the same network as SCL:
   "SysStart_Trigger" := "SysStart_Pb";
   "SysStop_Trigger" := "SysStop_Pb";
   "Sys_Running" := (("SysStart_Trigger" AND "AllHOAAuto") OR ("Sys_Running" AND NOT "SysStop_Trigger")) AND NOT "Critical_Alarm";
END_REGION
END_FUNCTION_BLOCK

FUNCTION_BLOCK "BACKWASH"   // FB7, LAD
{ S7_Optimized_Access := 'TRUE' }
VERSION : 0.1
   VAR
      ons1 : Bool;
      ons2 : Bool;
      ons3 : Bool;
      ons4 : Bool;
   END_VAR
   VAR_TEMP   // added for the SCL form of the ladder/FBD networks
      _w1 : Bool;
      _w2 : Bool;
      _w3 : Bool;
      _w4 : Bool;
   END_VAR
BEGIN

REGION Network 1
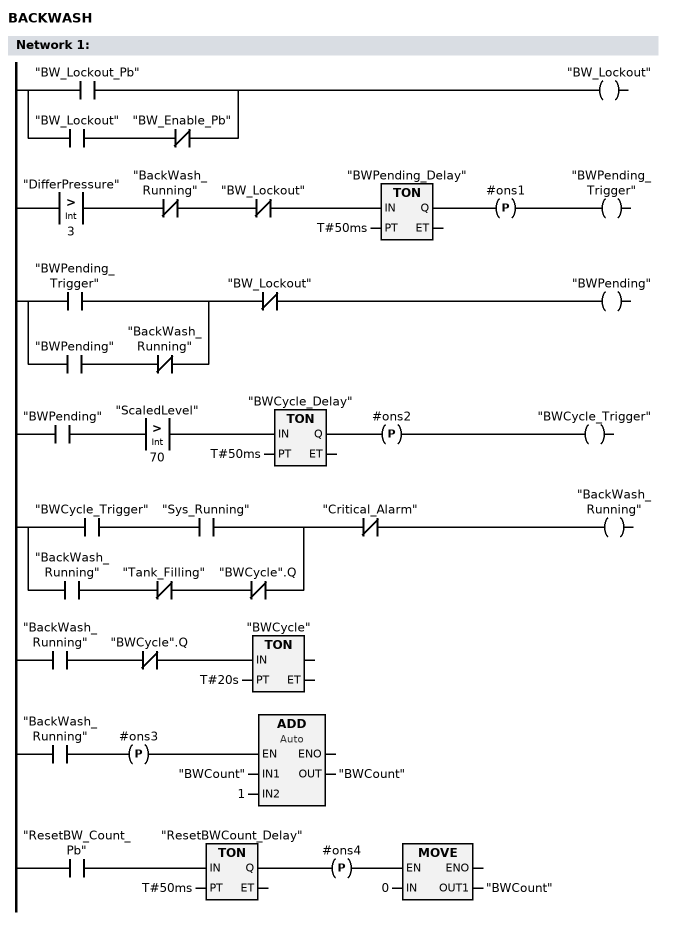
   "BW_Lockout" := "BW_Lockout_Pb" OR ("BW_Lockout" AND NOT "BW_Enable_Pb");
   "BWPending_Delay".TON(IN := ("DifferPressure" > 3) AND NOT "BackWash_Running" AND NOT "BW_Lockout",
                         PT := T#50ms);
   #_w1 := "BWPending_Delay".Q AND NOT #ons1;   // rising edge
   #ons1 := "BWPending_Delay".Q;
   "BWPending_Trigger" := #_w1;
   "BWPending" := ("BWPending_Trigger" OR ("BWPending" AND NOT "BackWash_Running")) AND NOT "BW_Lockout";
   "BWCycle_Delay".TON(IN := "BWPending" AND ("ScaledLevel" > 70), PT := T#50ms);
   #_w2 := "BWCycle_Delay".Q AND NOT #ons2;   // rising edge
   #ons2 := "BWCycle_Delay".Q;
   "BWCycle_Trigger" := #_w2;
   "BackWash_Running" := (("BWCycle_Trigger" AND "Sys_Running") OR ("BackWash_Running" AND NOT "Tank_Filling" AND NOT "BWCycle".Q)) AND NOT "Critical_Alarm";
   "BWCycle".TON(IN := "BackWash_Running" AND NOT "BWCycle".Q, PT := T#20s);
   #_w3 := "BackWash_Running" AND NOT #ons3;   // rising edge
   #ons3 := "BackWash_Running";
   IF #_w3 THEN "BWCount" := "BWCount" + 1; END_IF;
   "ResetBWCount_Delay".TON(IN := "ResetBW_Count_Pb", PT := T#50ms);
   #_w4 := "ResetBWCount_Delay".Q AND NOT #ons4;   // rising edge
   #ons4 := "ResetBWCount_Delay".Q;
   IF #_w4 THEN "BWCount" := 0; END_IF;
END_REGION
END_FUNCTION_BLOCK

FUNCTION_BLOCK "LEVEL"   // FB8, LAD
{ S7_Optimized_Access := 'TRUE' }
VERSION : 0.1
   VAR_TEMP   // added for the SCL form of the ladder/FBD networks
      _w1 : Bool;
      _w2 : Bool;
   END_VAR
BEGIN

REGION Network 1
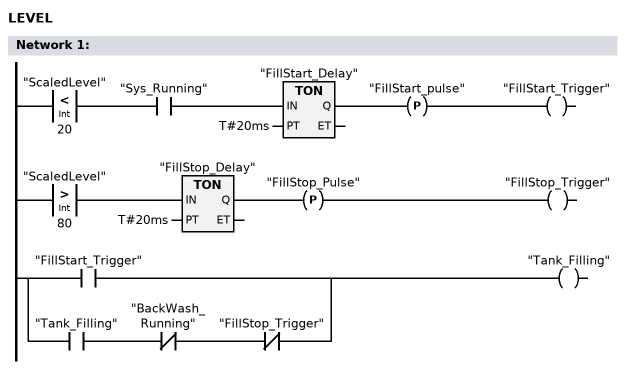
   "FillStart_Delay".TON(IN := ("ScaledLevel" < 20) AND "Sys_Running", PT := T#20ms);
   #_w1 := "FillStart_Delay".Q AND NOT "FillStart_pulse";   // rising edge
   "FillStart_pulse" := "FillStart_Delay".Q;
   "FillStart_Trigger" := #_w1;
   "FillStop_Delay".TON(IN := "ScaledLevel" > 80, PT := T#20ms);
   #_w2 := "FillStop_Delay".Q AND NOT "FillStop_Pulse";   // rising edge
   "FillStop_Pulse" := "FillStop_Delay".Q;
   "FillStop_Trigger" := #_w2;
   "Tank_Filling" := "FillStart_Trigger" OR ("Tank_Filling" AND NOT "BackWash_Running" AND NOT "FillStop_Trigger");
END_REGION
END_FUNCTION_BLOCK

FUNCTION_BLOCK "REVIEW"   // FB9, LAD
{ S7_Optimized_Access := 'TRUE' }
VERSION : 0.1
BEGIN

REGION Network 1
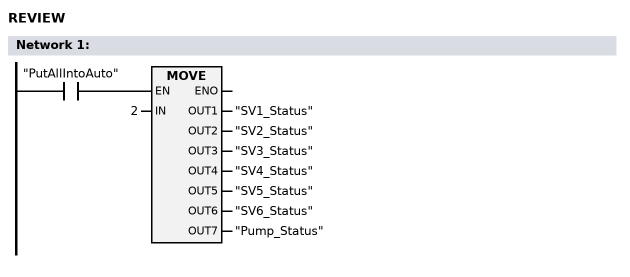
   RUNG wire#powerrail
      Contact( "PutAllIntoAuto" )
      { S7_GenerateENO := "TRUE" } Move(in := 2, out1 => "SV1_Status", out2 => "SV2_Status", out3 => "SV3_Status", out4 => "SV4_Status", out5 => "SV5_Status", out6 => "SV6_Status", out7 => "Pump_Status")
   END_RUNG
   // the same network as SCL:
   IF "PutAllIntoAuto" THEN
       "SV1_Status" := 2;
       "SV2_Status" := 2;
       "SV3_Status" := 2;
       "SV4_Status" := 2;
       "SV5_Status" := 2;
       "SV6_Status" := 2;
       "Pump_Status" := 2;
   END_IF;
END_REGION
END_FUNCTION_BLOCK

FUNCTION "Scaler" : Void   // FC1, FBD
{ S7_Optimized_Access := 'TRUE' }
VERSION : 0.1
   VAR_INPUT
      InputMin : Int;
      InputSignal : Int;
      InputMax : Int;
      ScaledMin : Int;
      ScaledMax : Int;
   END_VAR
   VAR_OUTPUT
      ScaledOut : Int;
   END_VAR
   VAR_TEMP
      tv : Real;
   END_VAR
BEGIN

REGION Network 1
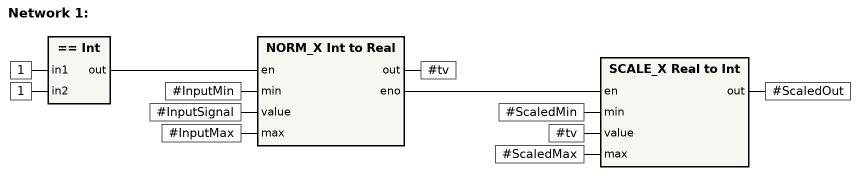
   // ENO of a box is taken as its EN; it also drops when the box reports an error
   IF 1 = 1 THEN
       #tv := NORM_X(MIN := #InputMin, VALUE := #InputSignal, MAX := #InputMax);
       #ScaledOut := SCALE_X(MIN := #ScaledMin, VALUE := #tv, MAX := #ScaledMax);
   END_IF;
END_REGION
END_FUNCTION

ORGANIZATION_BLOCK "Main"   // OB1, LAD, ProgramCycle
TITLE = "Main Program Sweep (Cycle)"
{ S7_Optimized_Access := 'TRUE' }
VERSION : 0.1
BEGIN

REGION Network 1
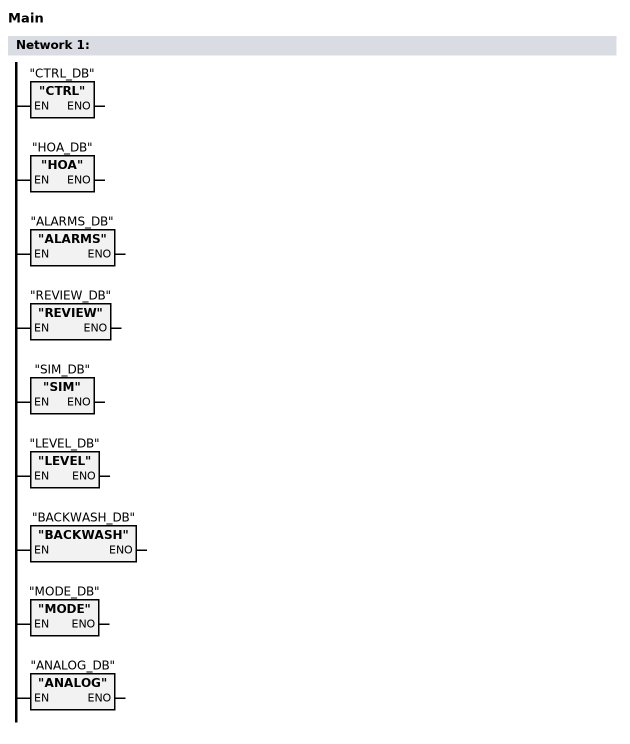
   RUNG wire#powerrail
      "CTRL_DB"()
   END_RUNG
   RUNG wire#powerrail
      "HOA_DB"()
   END_RUNG
   RUNG wire#powerrail
      "ALARMS_DB"()
   END_RUNG
   RUNG wire#powerrail
      "REVIEW_DB"()
   END_RUNG
   RUNG wire#powerrail
      "SIM_DB"()
   END_RUNG
   RUNG wire#powerrail
      "LEVEL_DB"()
   END_RUNG
   RUNG wire#powerrail
      "BACKWASH_DB"()
   END_RUNG
   RUNG wire#powerrail
      "MODE_DB"()
   END_RUNG
   RUNG wire#powerrail
      "ANALOG_DB"()
   END_RUNG
   // the same network as SCL:
   "CTRL_DB"();   // "CTRL"
   "HOA_DB"();   // "HOA"
   "ALARMS_DB"();   // "ALARMS"
   "REVIEW_DB"();   // "REVIEW"
   "SIM_DB"();   // "SIM"
   "LEVEL_DB"();   // "LEVEL"
   "BACKWASH_DB"();   // "BACKWASH"
   "MODE_DB"();   // "MODE"
   "ANALOG_DB"();   // "ANALOG"
END_REGION
END_ORGANIZATION_BLOCK

(* ===== HMI "HMI_RT_1" =====
system functions are stored by id; their names below are inferred from use
connection "PLC_1": S71200_TCP_IP, SCADA_S7_1200

HMI tags "Default tag table"
   "Solvalve1" : Bool = PLC SolValve1 AT %Q0.0, 500 ms
   "SolValve2" : Bool = PLC SolValve2 AT %Q0.1, 500 ms
   "Solvalve3" : Bool = PLC SolValve3 AT %Q0.2, 500 ms
   "Solvalve4" : Bool = PLC SolValve4 AT %Q0.3, 500 ms
   "SolValve5" : Bool = PLC SolValve5 AT %Q0.4, 500 ms
   "SolValve6" : Bool = PLC SolValve6 AT %Q0.5, 500 ms
   "Pump" : Bool = PLC Pump AT %Q0.6, 500 ms
   "ScaledLevel" : Int = PLC ScaledLevel AT %MW14, 500 ms
   "SysStart_Pb" : Bool = PLC SysStart_Pb AT %M32.1, 500 ms
   "DifferPressure" : Int = PLC DifferPressure AT %MW10, 500 ms
   "ScaledPressure1" : Int = PLC ScaledPressure1 AT %MW4, 500 ms
   "ScaledPressure2" : Int = PLC ScaledPressure2 AT %MW6, 500 ms
   "HiPres_Alarm" : Bool = PLC HiPres_Alarm AT %M34.3, 500 ms
   "LowFlow_Alarm" : Bool = PLC LowFlow_Alarm AT %M33.1, 500 ms
   "LowLevel_Alarm" : Bool = PLC LowLevel_Alarm AT %M33.4, 500 ms
   "HighLevel_Alarm" : Bool = PLC HighLevel_Alarm AT %M34.7, 500 ms
   "SysStop_Pb" : Bool = PLC SysStop_Pb AT %M32.5, 500 ms
   "Alarm_Reset" : Bool = PLC Alarm_Reset AT %M34.1, 500 ms
   "Alarm_Silence" : Bool = PLC Alarm_Silence AT %M34.5, 500 ms
   "HighLevelAlm_notify" : Bool = PLC HighLevelAlm_notify AT %M35.0, 500 ms
   "HiPres_Notify" : Bool = PLC HiPres_Notify AT %M34.4, 500 ms
   "LowAlarm_Notify" : Bool = PLC LowAlarm_Notify AT %M33.2, 500 ms
   "LowLevelAlm_Notify" : Bool = PLC LowLevelAlm_Notify AT %M33.5, 500 ms
   "FlowSwitch" : Bool = PLC FlowSwitch AT %M0.0, 500 ms
   "Tank_Filling" : Bool = PLC Tank_Filling AT %M39.0, 500 ms
   "Backwash_Running" : Bool = PLC BackWash_Running AT %M32.7, 500 ms
   "SV1Hand_Pb" : Bool = PLC SV1Hand_Pb AT %M16.1, 500 ms
   "SV1Off_Pb" : Bool = PLC SV1Off_Pb AT %M16.0, 500 ms
   "SV1Auto_Pb" : Bool = PLC SV1Auto_Pb AT %M16.2, 500 ms
   "SV2Hand_Pb" : Bool = PLC SV2Hand_Pb AT %M16.4, 500 ms
   "SV2Off_Pb" : Bool = PLC SV2Off_Pb AT %M16.3, 500 ms
   "SV2Auto_pb" : Bool = PLC SV2Auto_pb AT %M16.5, 500 ms
   "SV3Hand_pb" : Bool = PLC SV3Hand_pb AT %M16.7, 500 ms
   "SV3Off_pb" : Bool = PLC SV3Off_pb AT %M16.6, 500 ms
   "SV3Auto_Pb" : Bool = PLC SV3Auto_Pb AT %M17.0, 500 ms
   "SV4Hand_Pb" : Bool = PLC SV4Hand_Pb AT %M17.2, 500 ms
   "SV4Off_pb" : Bool = PLC SV4Off_pb AT %M17.1, 500 ms
   "SV4Auto_Pb" : Bool = PLC SV4Auto_Pb AT %M17.3, 500 ms
   "SV5Hand_Pb" : Bool = PLC SV5Hand_Pb AT %M17.5, 500 ms
   "SV5Off_Pb" : Bool = PLC SV5Off_Pb AT %M17.4, 500 ms
   "SV5Auto_Pb" : Bool = PLC SV5Auto_Pb AT %M17.6, 500 ms
   "SV6Hand_Pb" : Bool = PLC SV6Hand_Pb AT %M18.0, 500 ms
   "SV6Off_Pb" : Bool = PLC SV6Off_Pb AT %M17.7, 500 ms
   "SV6Auto_pb" : Bool = PLC SV6Auto_pb AT %M18.1, 500 ms
   "SV1_Status" : Int = PLC SV1_Status AT %MW18, 500 ms
   "SV2_Status" : Int = PLC SV2_Status AT %MW20, 500 ms
   "SV3_Status" : Int = PLC SV3_Status AT %MW22, 500 ms
   "SV4_Status" : Int = PLC SV4_Status AT %MW24, 500 ms
   "SV5_Status" : Int = PLC SV5_Status AT %MW26, 500 ms
   "SV6_Status" : Int = PLC SV6_Status AT %MW28, 500 ms
   "PumpHand_pb" : Bool = PLC PumpHand_pb AT %M2.1, 500 ms
   "PumpOff_pb" : Bool = PLC PumpOff_pb AT %M2.0, 500 ms
   "PumpAuto_pb" : Bool = PLC PumpAuto_pb AT %M2.2, 500 ms
   "Pump_Status" : Int = PLC Pump_Status AT %MW30, 500 ms

discrete alarms
   1: 'Tank level too high', class Errors, trigger "HighLevelAlm_notify" bit 0
   2: 'Pressure too high', class Errors, trigger "HiPres_Notify" bit 0
   3: 'No water flowing', class Errors, trigger "LowAlarm_Notify" bit 0
   4: 'Tank level too low', class Errors, trigger "LowLevelAlm_Notify" bit 0

screen "Schematic" 900x600
   TextField "Text field_1" at 330,13 size 240x28; Text 'SYSTEM SCHEMATIC'
   Bar "Bar_1" at 604,164 size 120x171; MinimumValue 0; MaximumValue 100
      ProcessValue <- "ScaledLevel"
   IOField "I/O field_1" at 410,289 size 39x20; FormatPattern s99999
      ProcessValue <- "DifferPressure"
   TubePolyline "Pipe_1" at 57,285 size 340x0
   TubePolyline "Pipe_2" at 458,283 size 147x0
   TubePolyline "Pipe_3" at 279,112 size 227x0
   TubePolyline "Pipe_4" at 147,453 size 376x0
   TubePolyline "Pipe_5" at 132,285 size 0x148
   TubePolyline "Pipe_6" at 537,328 size 0x113
   TubePolyline "Pipe_7" at 260,129 size 1x151
   TubePolyline "Pipe_8" at 524,129 size 0x154
   TubePolyline "Pipe_9" at 555,309 size 49x0
   TubePolyline "Pipe_10" at 236,358 size 93x0
   TubePolyline "Pipe_11" at 346,285 size 0x53
   TubeArcObject "Pipe elbow_1" at 256,108 size 23x24
   TubeArcObject "Pipe elbow_2" at 128,434 size 23x24
   TubeArcObject "Pipe elbow_3" at 518,433 size 23x24
   TubeArcObject "Pipe elbow_4" at 505,108 size 23x24
   TubeArcObject "Pipe elbow_5" at 533,305 size 23x24
   TubeArcObject "Pipe elbow_6" at 327,338 size 23x24
   TubePolyline "Pipe_12" at 724,294 size 49x0
   TubePolyline "Pipe_13" at 683,120 size 49x0
   TubeArcObject "Pipe elbow_7" at 660,116 size 23x24
   Button "Button_1" at 8,559 size 80x30; TextOff 'START'
      on PressLeft: SetBit("SysStart_Pb")
      on ReleaseLeft: ResetBit("SysStart_Pb")
   Button "Button_2" at 809,558 size 80x30; TextOff 'EXIT'
      on Click: StopRuntime(0)
   TextField "Text field_2" at 632,112 size 31x14; Text 'TANK'
   TextField "Text field_3" at 271,413 size 22x14; Text 'SV2'
   TextField "Text field_4" at 267,320 size 22x14; Text 'SV6'
   TextField "Text field_5" at 555,243 size 22x14; Text 'SV5'
   TextField "Text field_6" at 293,248 size 22x14; Text 'SV3'
   TextField "Text field_7" at 139,254 size 31x14; Text 'PUMP'
   TextField "Text field_8" at 76,248 size 22x14; Text 'SV1'
   TextField "Text field_9" at 337,76 size 22x14; Text 'SV4'
   IOField "I/O field_2" at 625,377 size 80x20; FormatPattern s99999
      ProcessValue <- "ScaledLevel"
   TextField "Text field_10" at 421,309 size 18x14; Text 'PSI'
   TextField "Text field_11" at 710,383 size 12x14; Text '%'
   TextField "Text field_12" at 406,140 size 38x14; Text 'FILTER'
   TextField "Text field_13" at 32,309 size 61x18; Text 'SUPPLY'
   TextField "Text field_14" at 773,302 size 66x18; Text 'TO USER'
   TextField "Text field_15" at 194,367 size 51x18; Text 'DRAIN'
   TextField "Text field_16" at 741,120 size 51x18; Text 'DRAIN'
   TextField "Text field_17" at 367,275 size 22x14; Text 'PT1'
   TextField "Text field_18" at 479,277 size 22x14; Text 'PT2'
   IOField "I/O field_3" at 355,304 size 34x25; FormatPattern s99999
      ProcessValue <- "ScaledPressure1"
   IOField "I/O field_4" at 472,304 size 34x25; FormatPattern s99999
      ProcessValue <- "ScaledPressure2"
   TextField "Text field_19" at 380,365 size 112x18; Text 'DIFFERENTIAL'
   TextField "Text field_20" at 381,383 size 81x18; Text 'PRESSURE'
   TextField "Text field_21" at 619,402 size 91x18; Text 'TANK LEVEL'
   Button "Button_3" at 95,559 size 80x30; TextOff 'STOP'
      on PressLeft: SetBit("SysStop_Pb")
      on ReleaseLeft: ResetBit("SysStop_Pb")
   Button "Button_4" at 496,558 size 80x30; TextOff 'ALARM'
      on Click: ActivateScreen("Alarm", 0)
   TextField "Text field_22" at 606,456 size 55x19; Text 'Alarm!!!'
   TextField "Text field_23" at 601,435 size 55x19; Text 'Alarm!!!'
   Line "Line_1" at 212,281 size 29x0
      Visibility <- "FlowSwitch"
   Line "Line_2" at 222,263 size 14x17
      Visibility <- "FlowSwitch"
   Group "Group" at 780,445 size 60x60
      Visibility <- "LowLevelAlm_Notify"
   Group "Group_1" at 780,445 size 60x60
      Visibility <- "HighLevelAlm_notify"
   Group "Group_2" at 780,445 size 60x60
      Visibility <- "HiPres_Notify"
   Group "Group_3" at 780,445 size 60x60
      Visibility <- "LowAlarm_Notify"
   TextField "Text field_28" at 201,291 size 56x14; Text 'FLOW SW'
   Button "Button_5" at 389,558 size 100x30; TextOff 'SECURITY'
      on Click: ActivateScreen("Security", 0)
   GraphicView "Graphic view_2" at 66,262 size 44x43; Picture "Graphic_22"
      Visibility <- "Solvalve1"
   GraphicView "Graphic view_1" at 66,263 size 44x42; Picture "Graphic_23"
      Visibility <- "Solvalve1"
   GraphicView "Graphic view_3" at 284,262 size 44x43; Picture "Graphic_22"
      Visibility <- "Solvalve3"
   GraphicView "Graphic view_4" at 545,257 size 44x43; Picture "Graphic_22"
      Visibility <- "SolValve5"
   GraphicView "Graphic view_5" at 260,429 size 44x43; Picture "Graphic_22"
      Visibility <- "SolValve2"
   GraphicView "Graphic view_6" at 257,335 size 44x43; Picture "Graphic_22"
      Visibility <- "SolValve6"
   GraphicView "Graphic view_7" at 327,90 size 44x43; Picture "Graphic_22"
      Visibility <- "Solvalve4"
   GraphicView "Graphic view_8" at 257,335 size 44x42; Picture "Graphic_23"
      Visibility <- "SolValve6"
   GraphicView "Graphic view_9" at 260,430 size 44x42; Picture "Graphic_23"
      Visibility <- "SolValve2"
   GraphicView "Graphic view_10" at 545,258 size 44x42; Picture "Graphic_23"
      Visibility <- "SolValve5"
   GraphicView "Graphic view_11" at 284,263 size 44x42; Picture "Graphic_23"
      Visibility <- "Solvalve3"
   GraphicView "Graphic view_12" at 327,90 size 44x42; Picture "Graphic_23"
      Visibility <- "Solvalve4"
   GraphicView "Graphic view_13" at 142,258 size 58x51; Picture "Graphic_20"
      Visibility <- "Pump"
   GraphicView "Graphic view_14" at 142,258 size 57x53; Picture "Graphic_25"
      Visibility <- "Pump"
   Polygon "Polygon_1" at 414,193 size 32x20
      Visibility <- "Tank_Filling"
   Polygon "Polygon_2" at 411,213 size 32x20
      Visibility <- "Backwash_Running"
   Button "Button_6" at 583,558 size 111x30; TextOff 'HOA CONFIG'
      on Click: ActivateScreen("HOAConfig", 0)
   Button "Button_7" at 701,558 size 100x30; TextOff 'TREND'
      on Click: ActivateScreen("Trend", 0)
   TextField "Text field_24" at 781,465 size 55x19; Text 'Alarm!!!'
   TextField "Text field_25" at 781,465 size 55x19; Text 'Alarm!!!'
   TextField "Text field_26" at 781,465 size 55x19; Text 'Alarm!!!'
   TextField "Text field_27" at 781,465 size 55x19; Text 'Alarm!!!'

screen "Alarm" 900x600
   TextField "Text field_1" at 359,13 size 183x28; Text 'ALARM SCREEN'
   AlarmControl "Alarm view_1" at 0,54 size 900x317
   Button "Button_2" at 813,558 size 80x30; TextOff 'EXIT'
      on Click: StopRuntime(0)
   Button "Button_4" at 367,558 size 111x30; TextOff 'SCHEMATIC'
      on Click: ActivateScreen("Schematic", 0)
   RoundButton "Round button_1" at 126,402 size 95x95; Text 'RESET'
      on PressLeft: SetBit("Alarm_Reset")
      on ReleaseLeft: ResetBit("Alarm_Reset")
   RoundButton "Round button_2" at 264,402 size 95x95; Text 'SILENCE'
      on PressLeft: SetBit("Alarm_Silence")
      on ReleaseLeft: ResetBit("Alarm_Silence")
   Button "Button_5" at 484,558 size 100x30; TextOff 'SECURITY'
      on Click: ActivateScreen("Alarm", 0)
      on Activate: ActivateScreen("Security", 0)
   Button "Button_6" at 590,558 size 111x30; TextOff 'HOA CONFIG'
      on Click: ActivateScreen("HOAConfig", 0)
   Button "Button_7" at 707,558 size 100x30; TextOff 'TREND'
      on Click: ActivateScreen("Trend", 0)

screen "Security" 800x600
   TextField "Text field_1" at 291,13 size 218x28; Text 'SECURITY SCREEN'
   UserView "User view_1" at 36,108 size 711x192
   Button "Button_1" at 192,376 size 119x50; TextOff 'LOG IN'
      on Click: function_a2a04561()
   Button "Button_2" at 353,376 size 119x50; TextOff 'LOG OUT'
   Group "Group" at 645,366 size 60x60
      Visibility <- "LowLevelAlm_Notify"
   Group "Group_1" at 645,366 size 60x60
      Visibility <- "HighLevelAlm_notify"
   Group "Group_2" at 645,366 size 60x60
      Visibility <- "HiPres_Notify"
   Group "Group_3" at 645,366 size 60x60
      Visibility <- "LowAlarm_Notify"
   Button "Button_4" at 271,557 size 111x30; TextOff 'SCHEMATIC'
      on Click: ActivateScreen("Schematic", 0)
   Button "Button_3" at 711,557 size 80x30; TextOff 'EXIT'
      on Click: StopRuntime(0)
   Button "Button_5" at 391,557 size 80x30; TextOff 'ALARM'
      on Click: ActivateScreen("Alarm", 0)
   Button "Button_6" at 481,557 size 111x30; TextOff 'HOA CONFIG'
      on Click: ActivateScreen("HOAConfig", 0)
   Button "Button_7" at 601,557 size 100x30; TextOff 'TREND'
      on Click: ActivateScreen("Trend", 0)
   TextField "Text field_24" at 646,386 size 55x19; Text 'Alarm!!!'
   TextField "Text field_25" at 646,386 size 55x19; Text 'Alarm!!!'
   TextField "Text field_26" at 646,386 size 55x19; Text 'Alarm!!!'
   TextField "Text field_27" at 646,386 size 55x19; Text 'Alarm!!!'

screen "HOAConfig" 900x600
   TextField "Text field_1" at 330,13 size 262x28; Text 'HOA CONFIGURATION'
   Button "Button_2" at 809,559 size 80x30; TextOff 'EXIT'
      on Click: StopRuntime(0)
   Button "Button_4" at 390,559 size 111x30; TextOff 'SCHEMATIC'
      on Click: ActivateScreen("Schematic", 0)
   Button "Button_5" at 508,559 size 100x30; TextOff 'SECURITY'
      on Click: ActivateScreen("Alarm", 0)
      on Activate: ActivateScreen("Security", 0)
   Button "Button_1" at 722,559 size 80x30; TextOff 'ALARM'
      on Click: ActivateScreen("Alarm", 0)
   Button "Button_3" at 552,341 size 45x30; TextOff 'H'
      on PressLeft: SetBit("PumpHand_pb")
      on ReleaseLeft: ResetBit("PumpHand_pb")
   Button "Button_6" at 271,315 size 45x30; TextOff 'O'
      on PressLeft: SetBit("SV4Off_pb")
      on ReleaseLeft: ResetBit("SV4Off_pb")
   Button "Button_7" at 215,315 size 45x30; TextOff 'H'
      on PressLeft: SetBit("SV4Hand_Pb")
      on ReleaseLeft: ResetBit("SV4Hand_Pb")
   Button "Button_8" at 271,274 size 45x30; TextOff 'O'
      on PressLeft: SetBit("SV3Off_pb")
      on ReleaseLeft: ResetBit("SV3Off_pb")
   Button "Button_9" at 271,236 size 45x30; TextOff 'O'
      on PressLeft: SetBit("SV2Off_Pb")
      on ReleaseLeft: ResetBit("SV2Off_Pb")
   Button "Button_10" at 215,274 size 45x30; TextOff 'H'
      on PressLeft: SetBit("SV3Hand_pb")
      on ReleaseLeft: ResetBit("SV3Hand_pb")
   Button "Button_11" at 215,236 size 45x30; TextOff 'H'
      on PressLeft: SetBit("SV2Hand_Pb")
      on ReleaseLeft: ResetBit("SV2Hand_Pb")
   Button "Button_12" at 325,192 size 45x30; TextOff 'A'
      on PressLeft: SetBit("SV1Auto_Pb")
      on ReleaseLeft: ResetBit("SV1Auto_Pb")
   Button "Button_13" at 215,192 size 45x30; TextOff 'H'
      on PressLeft: SetBit("SV1Hand_Pb")
      on ReleaseLeft: ResetBit("SV1Hand_Pb")
   Button "Button_14" at 325,236 size 45x30; TextOff 'A'
      on PressLeft: SetBit("SV2Auto_pb")
      on ReleaseLeft: ResetBit("SV2Auto_pb")
   Button "Button_15" at 271,192 size 45x30; TextOff 'O'
      on PressLeft: SetBit("SV1Off_Pb")
      on ReleaseLeft: ResetBit("SV1Off_Pb")
   Button "Button_16" at 325,315 size 45x30; TextOff 'A'
      on PressLeft: SetBit("SV4Auto_Pb")
      on ReleaseLeft: ResetBit("SV4Auto_Pb")
   Button "Button_18" at 608,341 size 45x30; TextOff 'O'
      on PressLeft: SetBit("PumpOff_pb")
      on ReleaseLeft: ResetBit("PumpOff_pb")
   Button "Button_19" at 664,341 size 45x30; TextOff 'A'
      on PressLeft: SetBit("PumpAuto_pb")
      on ReleaseLeft: ResetBit("PumpAuto_pb")
   Button "Button_20" at 325,399 size 45x30; TextOff 'A'
      on PressLeft: SetBit("SV6Auto_pb")
      on ReleaseLeft: ResetBit("SV6Auto_pb")
   Button "Button_21" at 271,399 size 45x30; TextOff 'O'
      on PressLeft: SetBit("SV6Off_Pb")
      on ReleaseLeft: ResetBit("SV6Off_Pb")
   Button "Button_22" at 215,399 size 45x30; TextOff 'H'
      on PressLeft: SetBit("SV6Hand_Pb")
      on ReleaseLeft: ResetBit("SV6Hand_Pb")
   Button "Button_23" at 325,356 size 46x30; TextOff 'A'
      on PressLeft: SetBit("SV5Auto_Pb")
      on ReleaseLeft: ResetBit("SV5Auto_Pb")
   Button "Button_24" at 325,274 size 45x30; TextOff 'A'
      on PressLeft: SetBit("SV3Auto_Pb")
      on ReleaseLeft: ResetBit("SV3Auto_Pb")
   Button "Button_25" at 271,357 size 45x30; TextOff 'O'
      on PressLeft: SetBit("SV5Off_Pb")
      on ReleaseLeft: ResetBit("SV5Off_Pb")
   Button "Button_26" at 215,357 size 45x30; TextOff 'H'
      on PressLeft: SetBit("SV5Hand_Pb")
      on ReleaseLeft: ResetBit("SV5Hand_Pb")
   TextField "Text field_16" at 138,200 size 58x18; Text 'VALVE1'
   TextField "Text field_2" at 138,282 size 58x18; Text 'VALVE3'
   TextField "Text field_3" at 138,323 size 58x18; Text 'VALVE4'
   TextField "Text field_4" at 138,368 size 58x18; Text 'VALVE5'
   TextField "Text field_5" at 138,411 size 58x18; Text 'VALVE6'
   TextField "Text field_6" at 138,244 size 58x18; Text 'VALVE2'
   TextField "Text field_7" at 606,301 size 55x23; Text 'PUMP'
   Circle "Circle_1" at 391,194 size 31x31
      Appearance <- "SV1_Status"
   Circle "Circle_2" at 391,233 size 31x31
      Appearance <- "SV2_Status"
   Circle "Circle_3" at 390,276 size 31x31
      Appearance <- "SV3_Status"
   Circle "Circle_4" at 390,316 size 31x31
      Appearance <- "SV4_Status"
   Circle "Circle_5" at 390,357 size 31x31
      Appearance <- "SV5_Status"
   Circle "Circle_6" at 390,400 size 31x31
      Appearance <- "SV6_Status"
   Circle "Circle_7" at 736,340 size 31x31
      Appearance <- "Pump_Status"
   Button "Button_17" at 615,559 size 100x30; TextOff 'TREND'
      on Click: ActivateScreen("Trend", 0)
   TextField "Text field_8" at 198,143 size 189x23; Text 'SOLENOID VALVES'
   TextField "Text field_9" at 557,190 size 11x19; Text 'H'
   TextField "Text field_11" at 557,256 size 11x19; Text 'A'
   TextField "Text field_10" at 556,222 size 12x19; Text 'O'
   TextField "Text field_12" at 595,194 size 44x18; Text 'HAND'
   TextField "Text field_13" at 596,222 size 30x18; Text 'OFF'
   TextField "Text field_14" at 596,256 size 42x18; Text 'AUTO'

screen "Trend" 900x600
   TextField "Text field_1" at 410,13 size 80x28; Text 'TREND'
   Button "Button_2" at 809,559 size 80x30; TextOff 'EXIT'
      on Click: StopRuntime(0)
   Button "Button_4" at 607,559 size 80x30; TextOff 'ALARM'
      on Click: ActivateScreen("Alarm", 0)
   Button "Button_5" at 501,559 size 100x30; TextOff 'SECURITY'
      on Click: ActivateScreen("Alarm", 0)
      on Activate: ActivateScreen("Security", 0)
   Button "Button_6" at 692,559 size 111x30; TextOff 'HOA CONFIG'
      on Click: ActivateScreen("HOAConfig", 0)
   Button "Button_1" at 383,559 size 111x30; TextOff 'SCHEMATIC'
      on Click: ActivateScreen("Schematic", 0)
   OnlineTrendControl "f(t) trend view_1" at 28,71 size 857x420
*)